INTERFACE I_MotionInterlocksLimSw EXTENDS I_MotionInterlocks

PROPERTY LimHit : BOOL
GET
END_GET
END_PROPERTY

PROPERTY LimHitIdling : BOOL
GET
END_GET
END_PROPERTY

PROPERTY LimHitMoving : BOOL
GET
END_GET
END_PROPERTY

END_INTERFACE

(* stored: Version 1.1.0.1
   Itf I_MotionInterlocksLimSw: Id {e002b16f-1804-418d-93ce-ce168a098275}
   Property LimHit: Id {00f31b83-20b0-4e18-bb57-b84a58adcd1b}
   Get Get: Id {dc48a399-6ef3-4f49-9589-4858181b8029}
   Property LimHitIdling: Id {a9898372-986c-4ee4-bc98-43640fd003f2}
   Get Get: Id {d9233391-3505-4407-ade5-ca790ab05516}
   Property LimHitMoving: Id {12768a8b-8e2d-462d-ac59-05ed276cdf42}
   Get Get: Id {f40fa498-6562-48ff-8455-7f34f6bbcf01} *)
